TYPE EventTestsystem :
STRUCT
  logging: EventRunner;
  event: Event := (logging:=logging);
END_STRUCT
END_TYPE

(* stored: Version 1.1.0.1, ProductVersion 3.1.4024.9
   DUT EventTestsystem: Id {1d1d3ef4-d20e-433d-90eb-bc663d6abd18} *)
